PROGRAM MAIN
VAR
	myVeryFirstTcoContextInstance :	TcoContext;
END_VAR

myVeryFirstTcoContextInstance.Run();

END_PROGRAM

(* stored: Version 1.1.0.1, ProductVersion 3.1.4024.11
   POU MAIN: Id {9359a558-9122-0f04-2d2f-c4fb3f11651d}, SpecialFunc None *)
